{attribute 'pack_mode' := '1'}
TYPE ClearAxisFaults EXTENDS IncomingMessage :
STRUCT
	axisIndex: INT; (* 1 or 2.*)
END_STRUCT
END_TYPE

(* stored: Version 1.1.0.1, ProductVersion 3.1.4022.12
   DUT ClearAxisFaults: Id {1546c464-a4ba-4de2-ac55-bf0b9dc631d2} *)
